PROGRAM SafetyHandling
VAR
	restart_safety 	: TP;
	//safety_state 	: RS;
	start_delay 	: TON;
	ErrAck_Pulse	: TP;
	//SafetyLog		: FB_EventLog;
	Run:		BOOL := TRUE;
	Restart:	BOOL;
	ErrAck:		BOOL;
END_VAR
VAR_OUTPUT
	Error:	BOOL;
	Stop:	BOOL;
END_VAR

// Safety can be stopped by pressing STOP and RESET on main panel
GVL_Safety.Run := Run;
// power on delay for Safety RESTART after RUN=1
restart_safety(IN := TRUE, PT := T#1S);
// RESTART Safety after pushing reset or power on delay
// GVL_Safety.Restart := restart_safety.Q;
GVL_Safety.Restart := Restart;
// wait n seconds after Start ...
start_delay(IN := TRUE, PT := T#2S);
// ... and send ErrAck for n milliseconds
ErrAck_Pulse(IN := start_delay.Q, PT := T#200MS);

// Error Acknowledgment: Turn key_switch OFF and press STOP 
// GVL_Safety.ErrAck := ErrAck_Pulse.Q;
GVL_Safety.ErrAck := ErrAck;
Stop := GVL_Safety.Stop;
Error := GVL_Safety.Error;


//SafetyLog(Trigger := Error,
//				Level := ADSLOG_MSGTYPE_ERROR,
//				OnMessage := 'Safety Error! Emergency stop enganged!',
//				OffMessage := 'Safety is OK.',
//				OffLevel := ADSLOG_MSGTYPE_HINT);

END_PROGRAM

(* stored: Version 1.1.0.1, ProductVersion 3.1.4024.9
   POU SafetyHandling: Id {6d4a788c-2168-4769-93de-c67314036861}, SpecialFunc None *)
